// TIA Portal V20 export
ORGANIZATION_BLOCK "CyclicInterrupt_1"   // OB30, LAD, CyclicInterrupt
{ S7_Optimized_Access := 'TRUE' }
// stored: SetENOAutomatically false
BEGIN
END_ORGANIZATION_BLOCK
